Staubli VAL3: getTrajType.pgx

program getTrajType(string& x_sTrajType[] (dimensions=1))
  local num l_nPos
  local string l_sPath
begin
  // get the trajType
  l_sPath=libPath()
  if find(l_sPath,sTrajType)==-1 or sTrajType==""
    do
      l_nPos=find(l_sPath,"/")
      if l_nPos==-1
        l_nPos=find(l_sPath,"\")
      endIf
      if l_nPos!=-1
        l_sPath=right(l_sPath,len(l_sPath)-l_nPos-1)
      endIf
    until l_nPos==-1
    //
    sTrajType=l_sPath
  endIf
  // return back
  x_sTrajType=sTrajType
end
